LIN {X 0,Y 82.914,Z 593.303,A -85,B 0,C 180,E1 -30407.099,E2 -30407.099} C_VEL
LIN {X 0,Y 91.318,Z 585.109,A -85,B 0,C 180,E1 -30408.889,E2 -30408.889} C_VEL
LIN {X 0,Y 99.802,Z 575.115,A -85,B 0,C 180,E1 -30410.355,E2 -30410.355} C_VEL
LIN {X 0,Y 107.491,Z 563.809,A -85,B 0,C 180,E1 -30411.456,E2 -30411.456} C_VEL
LIN {X 0,Y 114.033,Z 551.61,A -85,B 0,C 180,E1 -30412.293,E2 -30412.293} C_VEL
LIN {X 0,Y 119.005,Z 539.43,A -85,B 0,C 180,E1 -30412.792,E2 -30412.792} C_VEL
LIN {X 0,Y 122.619,Z 526.994,A -85,B 0,C 180,E1 -30413.207,E2 -30413.207} C_VEL
LIN {X 0,Y 122.694,Z 526.451,A -85,B 0,C 180,E1 -30413.422,E2 -30413.422} C_VEL
LIN {X 0,Y 122.556,Z 525.141,A -85,B 0,C 180,E1 -30415.478,E2 -30415.478} C_VEL
LIN {X 0,Y 122.565,Z 523.201,A -85,B 0,C 180,E1 -30420,E2 -30420} C_VEL
LIN {X 0,Y 122.551,Z 525.424,A -85,B 0,C 180,E1 -30425.554,E2 -30425.554} C_VEL
LIN {X 0,Y 122.631,Z 526.514,A -85,B 0,C 180,E1 -30427.085,E2 -30427.085} C_VEL
LIN {X 0,Y 119.046,Z 538.887,A -85,B 0,C 180,E1 -30427.632,E2 -30427.632} C_VEL
LIN {X 0,Y 114.177,Z 550.868,A -85,B 0,C 180,E1 -30428.279,E2 -30428.279} C_VEL
LIN {X 0,Y 107.695,Z 563.005,A -85,B 0,C 180,E1 -30429.238,E2 -30429.238} C_VEL
LIN {X 0,Y 100.063,Z 574.276,A -85,B 0,C 180,E1 -30430.489,E2 -30430.489} C_VEL
LIN {X 0,Y 91.356,Z 584.529,A -85,B 0,C 180,E1 -30432.152,E2 -30432.152} C_VEL
LIN {X 0,Y 87.175,Z 588.67,A -85,B 0,C 180,E1 -30432.621,E2 -30432.621} C_VEL
LIN {X 0,Y 79.586,Z 595.067,A -85,B 0,C 180,E1 -30432.363,E2 -30432.363} C_VEL
LIN {X 0,Y 71.531,Z 600.835,A -85,B 0,C 180,E1 -30432.172,E2 -30432.172} C_VEL
LIN {X 0,Y 66.625,Z 603.967,A -85,B 0,C 180,E1 -30432.991,E2 -30432.991} C_VEL
LIN {X 0,Y 58.426,Z 608.742,A -85,B 0,C 180,E1 -30435.785,E2 -30435.785} C_VEL
LIN {X 0,Y 48.676,Z 613.433,A -85,B 0,C 180,E1 -30440.205,E2 -30440.205} C_VEL
LIN {X 0,Y 39.401,Z 617.015,A -85,B 0,C 180,E1 -30446.896,E2 -30446.896} C_VEL
LIN {X 0,Y 33.637,Z 618.862,A -85,B 0,C 180,E1 -30453.309,E2 -30453.309} C_VEL
LIN {X 0,Y 28.389,Z 620.248,A -85,B 0,C 180,E1 -30462.044,E2 -30462.044} C_VEL
LIN {X 0,Y 21.1,Z 621.833,A -85,B 0,C 180,E1 -30490.548,E2 -30490.548} C_VEL
LIN {X 0,Y 20.153,Z 622.053,A -85,B 0,C 180,E1 -30510.004,E2 -30510.004} C_VEL
LIN {X 0,Y 21.101,Z 621.857,A -85,B 0,C 180,E1 -30529.459,E2 -30529.459} C_VEL
LIN {X 0,Y 28.389,Z 620.301,A -85,B 0,C 180,E1 -30557.964,E2 -30557.964} C_VEL
LIN {X 0,Y 33.629,Z 618.939,A -85,B 0,C 180,E1 -30566.718,E2 -30566.718} C_VEL
LIN {X 0,Y 42.388,Z 616.065,A -85,B 0,C 180,E1 -30575.777,E2 -30575.777} C_VEL
LIN {X 0,Y 51.868,Z 612.161,A -85,B 0,C 180,E1 -30581.536,E2 -30581.536} C_VEL
LIN {X 0,Y 61.711,Z 607.122,A -85,B 0,C 180,E1 -30585.478,E2 -30585.478} C_VEL
LIN {X 0,Y 71.724,Z 600.776,A -85,B 0,C 180,E1 -30588.489,E2 -30588.489} C_VEL
LIN {X 0,Y 81.857,Z 592.844,A -85,B 0,C 180,E1 -30590.889,E2 -30590.889} C_VEL
LIN {X 0,Y 90.404,Z 584.751,A -85,B 0,C 180,E1 -30592.397,E2 -30592.397} C_VEL
LIN {X 0,Y 99.006,Z 574.873,A -85,B 0,C 180,E1 -30593.627,E2 -30593.627} C_VEL
LIN {X 0,Y 105.908,Z 565.141,A -85,B 0,C 180,E1 -30594.508,E2 -30594.508} C_VEL
LIN {X 0,Y 111.969,Z 554.581,A -85,B 0,C 180,E1 -30595.174,E2 -30595.174} C_VEL
LIN {X 0,Y 117.484,Z 542.178,A -85,B 0,C 180,E1 -30595.75,E2 -30595.75} C_VEL
LIN {X 0,Y 120.918,Z 531.884,A -85,B 0,C 180,E1 -30596.19,E2 -30596.19} C_VEL
LIN {X 0,Y 121.07,Z 530.606,A -85,B 0,C 180,E1 -30600,E2 -30600} C_VEL
LIN {X 0,Y 120.958,Z 531.95,A -85,B 0,C 180,E1 -30603.518,E2 -30603.518} C_VEL
LIN {X 0,Y 116.623,Z 544.629,A -85,B 0,C 180,E1 -30603.898,E2 -30603.898} C_VEL
LIN {X 0,Y 111.022,Z 556.642,A -85,B 0,C 180,E1 -30604.412,E2 -30604.412} C_VEL
LIN {X 0,Y 104.067,Z 568.172,A -85,B 0,C 180,E1 -30605.036,E2 -30605.036} C_VEL
LIN {X 0,Y 96.264,Z 578.56,A -85,B 0,C 180,E1 -30605.873,E2 -30605.873} C_VEL
LIN {X 0,Y 88.501,Z 587.056,A -85,B 0,C 180,E1 -30606.943,E2 -30606.943} C_VEL
LIN {X 0,Y 78.201,Z 596.263,A -85,B 0,C 180,E1 -30608.658,E2 -30608.658} C_VEL
LIN {X 0,Y 68.017,Z 603.672,A -85,B 0,C 180,E1 -30610.998,E2 -30610.998} C_VEL
LIN {X 0,Y 58.02,Z 609.627,A -85,B 0,C 180,E1 -30614.286,E2 -30614.286} C_VEL
LIN {X 0,Y 48.239,Z 614.33,A -85,B 0,C 180,E1 -30618.732,E2 -30618.732} C_VEL
LIN {X 0,Y 38.876,Z 617.925,A -85,B 0,C 180,E1 -30625.32,E2 -30625.32} C_VEL
LIN {X 0,Y 33.022,Z 619.778,A -85,B 0,C 180,E1 -30631.64,E2 -30631.64} C_VEL
LIN {X 0,Y 23.519,Z 622.171,A -85,B 0,C 180,E1 -30653.294,E2 -30653.294} C_VEL
LIN {X 0,Y 20.748,Z 622.783,A -85,B 0,C 180,E1 -30670.196,E2 -30670.196} C_VEL
LIN {X 0,Y 19.968,Z 622.998,A -85,B 0,C 180,E1 -30689.996,E2 -30689.996} C_VEL
LIN {X 0,Y 20.747,Z 622.762,A -85,B 0,C 180,E1 -30709.797,E2 -30709.797} C_VEL
LIN {X 0,Y 27.808,Z 621.124,A -85,B 0,C 180,E1 -30739.302,E2 -30739.302} C_VEL
LIN {X 0,Y 33.019,Z 619.708,A -85,B 0,C 180,E1 -30748.36,E2 -30748.36} C_VEL
LIN {X 0,Y 41.939,Z 616.756,A -85,B 0,C 180,E1 -30757.169,E2 -30757.169} C_VEL
LIN {X 0,Y 51.476,Z 612.766,A -85,B 0,C 180,E1 -30762.879,E2 -30762.879} C_VEL
LIN {X 0,Y 62.803,Z 606.729,A -85,B 0,C 180,E1 -30767.517,E2 -30767.517} C_VEL
LIN {X 0,Y 73.089,Z 599.938,A -85,B 0,C 180,E1 -30770.264,E2 -30770.264} C_VEL
LIN {X 0,Y 83.334,Z 591.643,A -85,B 0,C 180,E1 -30772.275,E2 -30772.275} C_VEL
LIN {X 0,Y 91.939,Z 583.13,A -85,B 0,C 180,E1 -30773.584,E2 -30773.584} C_VEL
LIN {X 0,Y 100.593,Z 572.617,A -85,B 0,C 180,E1 -30774.613,E2 -30774.613} C_VEL
LIN {X 0,Y 107.539,Z 562.211,A -85,B 0,C 180,E1 -30775.296,E2 -30775.296} C_VEL
LIN {X 0,Y 113.652,Z 550.719,A -85,B 0,C 180,E1 -30775.865,E2 -30775.865} C_VEL
LIN {X 0,Y 118.471,Z 538.818,A -85,B 0,C 180,E1 -30776.212,E2 -30776.212} C_VEL
LIN {X 0,Y 120.685,Z 531.737,A -85,B 0,C 180,E1 -30776.469,E2 -30776.469} C_VEL
LIN {X 0,Y 120.828,Z 530.26,A -85,B 0,C 180,E1 -30780,E2 -30780} C_VEL
LIN {X 0,Y 120.635,Z 531.717,A -85,B 0,C 180,E1 -30783.953,E2 -30783.953} C_VEL
LIN {X 0,Y 116.344,Z 544.263,A -85,B 0,C 180,E1 -30784.417,E2 -30784.417} C_VEL
LIN {X 0,Y 111.109,Z 555.609,A -85,B 0,C 180,E1 -30784.978,E2 -30784.978} C_VEL
LIN {X 0,Y 104.189,Z 567.217,A -85,B 0,C 180,E1 -30785.766,E2 -30785.766} C_VEL
LIN {X 0,Y 96.43,Z 577.65,A -85,B 0,C 180,E1 -30786.78,E2 -30786.78} C_VEL
LIN {X 0,Y 88.707,Z 586.174,A -85,B 0,C 180,E1 -30787.973,E2 -30787.973} C_VEL
LIN {X 0,Y 80.169,Z 594.029,A -85,B 0,C 180,E1 -30789.523,E2 -30789.523} C_VEL
LIN {X 0,Y 70.069,Z 601.693,A -85,B 0,C 180,E1 -30792.06,E2 -30792.06} C_VEL
LIN {X 0,Y 66.625,Z 603.967,A -85,B 0,C 180,E1 -30792.991,E2 -30792.991} C_VEL
LIN {X 0,Y 61.58,Z 606.937,A -85,B 0,C 180,E1 -30793.946,E2 -30793.946} C_VEL
LIN {X 0,Y 52.651,Z 611.259,A -85,B 0,C 180,E1 -30794.024,E2 -30794.024} C_VEL
LIN {X 0,Y 43.448,Z 614.93,A -85,B 0,C 180,E1 -30794.239,E2 -30794.239} C_VEL
LIN {X 0,Y 38.01,Z 616.77,A -85,B 0,C 180,E1 -30796.127,E2 -30796.127} C_VEL
LIN {X 0,Y 30.317,Z 619.031,A -85,B 0,C 180,E1 -30801.995,E2 -30801.995} C_VEL
LIN {X 0,Y 24.208,Z 620.416,A -85,B 0,C 180,E1 -30809.435,E2 -30809.435} C_VEL
LIN {X 0,Y 14.59,Z 622.001,A -85,B 0,C 180,E1 -30841.21,E2 -30841.21} C_VEL
LIN {X 0,Y 13.051,Z 622.22,A -85,B 0,C 180,E1 -30870.006,E2 -30870.006} C_VEL
LIN {X 0,Y 14.592,Z 622.024,A -85,B 0,C 180,E1 -30898.799,E2 -30898.799} C_VEL
LIN {X 0,Y 24.208,Z 620.468,A -85,B 0,C 180,E1 -30930.576,E2 -30930.576} C_VEL
LIN {X 0,Y 30.312,Z 619.106,A -85,B 0,C 180,E1 -30938.043,E2 -30938.043} C_VEL
LIN {X 0,Y 39.999,Z 616.232,A -85,B 0,C 180,E1 -30945.111,E2 -30945.111} C_VEL
LIN {X 0,Y 50.073,Z 612.327,A -85,B 0,C 180,E1 -30949.271,E2 -30949.271} C_VEL
LIN {X 0,Y 60.322,Z 607.288,A -85,B 0,C 180,E1 -30952.033,E2 -30952.033} C_VEL
LIN {X 0,Y 71.596,Z 600.267,A -85,B 0,C 180,E1 -30954.366,E2 -30954.366} C_VEL
LIN {X 0,Y 81.035,Z 593.009,A -85,B 0,C 180,E1 -30955.859,E2 -30955.859} C_VEL
LIN {X 0,Y 89.741,Z 584.915,A -85,B 0,C 180,E1 -30956.896,E2 -30956.896} C_VEL
LIN {X 0,Y 98.471,Z 575.036,A -85,B 0,C 180,E1 -30957.728,E2 -30957.728} C_VEL
LIN {X 0,Y 106.343,Z 563.897,A -85,B 0,C 180,E1 -30958.379,E2 -30958.379} C_VEL
LIN {X 0,Y 113.154,Z 551.609,A -85,B 0,C 180,E1 -30958.922,E2 -30958.922} C_VEL
LIN {X 0,Y 118.05,Z 540.074,A -85,B 0,C 180,E1 -30959.253,E2 -30959.253} C_VEL
LIN {X 0,Y 118.638,Z 538.372,A -85,B 0,C 180,E1 -30959.307,E2 -30959.307} C_VEL
LIN {X 0,Y 118.938,Z 537.482,A -85,B 0,C 180,E1 -30959.577,E2 -30959.577} C_VEL
LIN {X 0,Y 118.928,Z 537.521,A -85,B 0,C 180,E1 -30960,E2 -30960} C_VEL
LIN {X 0,Y 118.663,Z 538.323,A -85,B 0,C 180,E1 -30960.282,E2 -30960.282} C_VEL
LIN {X 0,Y 113.841,Z 550.25,A -85,B 0,C 180,E1 -30960.588,E2 -30960.588} C_VEL
LIN {X 0,Y 107.194,Z 562.581,A -85,B 0,C 180,E1 -30960.947,E2 -30960.947} C_VEL
LIN {X 0,Y 99.302,Z 574.069,A -85,B 0,C 180,E1 -30961.403,E2 -30961.403} C_VEL
LIN {X 0,Y 91.421,Z 583.316,A -85,B 0,C 180,E1 -30961.99,E2 -30961.99} C_VEL
LIN {X 0,Y 82.683,Z 591.755,A -85,B 0,C 180,E1 -30962.849,E2 -30962.849} C_VEL
LIN {X 0,Y 72.229,Z 600,A -85,B 0,C 180,E1 -30964.16,E2 -30964.16} C_VEL
LIN {X 0,Y 61.837,Z 606.651,A -85,B 0,C 180,E1 -30966.029,E2 -30966.029} C_VEL
LIN {X 0,Y 49.851,Z 612.733,A -85,B 0,C 180,E1 -30969.29,E2 -30969.29} C_VEL
LIN {X 0,Y 39.724,Z 616.687,A -85,B 0,C 180,E1 -30973.319,E2 -30973.319} C_VEL
LIN {X 0,Y 29.904,Z 619.611,A -85,B 0,C 180,E1 -30979.926,E2 -30979.926} C_VEL
LIN {X 0,Y 18.315,Z 622.004,A -85,B 0,C 180,E1 -30999.865,E2 -30999.865} C_VEL
LIN {X 0,Y 14.253,Z 622.616,A -85,B 0,C 180,E1 -31020.449,E2 -31020.449} C_VEL
LIN {X 0,Y 12.865,Z 622.83,A -85,B 0,C 180,E1 -31049.994,E2 -31049.994} C_VEL
LIN {X 0,Y 14.252,Z 622.594,A -85,B 0,C 180,E1 -31079.541,E2 -31079.541} C_VEL
LIN {X 0,Y 23.783,Z 620.956,A -85,B 0,C 180,E1 -31112.434,E2 -31112.434} C_VEL
LIN {X 0,Y 29.901,Z 619.54,A -85,B 0,C 180,E1 -31120.075,E2 -31120.075} C_VEL
LIN {X 0,Y 39.721,Z 616.587,A -85,B 0,C 180,E1 -31126.684,E2 -31126.684} C_VEL
LIN {X 0,Y 49.847,Z 612.597,A -85,B 0,C 180,E1 -31130.722,E2 -31130.722} C_VEL
LIN {X 0,Y 61.656,Z 606.56,A -85,B 0,C 180,E1 -31133.997,E2 -31133.997} C_VEL
LIN {X 0,Y 72.226,Z 599.768,A -85,B 0,C 180,E1 -31135.84,E2 -31135.84} C_VEL
LIN {X 0,Y 82.679,Z 591.474,A -85,B 0,C 180,E1 -31137.166,E2 -31137.166} C_VEL
LIN {X 0,Y 91.418,Z 582.96,A -85,B 0,C 180,E1 -31138.019,E2 -31138.019} C_VEL
LIN {X 0,Y 100.175,Z 572.446,A -85,B 0,C 180,E1 -31138.668,E2 -31138.668} C_VEL
LIN {X 0,Y 108.067,Z 560.606,A -85,B 0,C 180,E1 -31139.13,E2 -31139.13} C_VEL
LIN {X 0,Y 113.978,Z 549.173,A -85,B 0,C 180,E1 -31139.487,E2 -31139.487} C_VEL
LIN {X 0,Y 118.388,Z 538.126,A -85,B 0,C 180,E1 -31139.661,E2 -31139.661} C_VEL
LIN {X 0,Y 118.698,Z 537.187,A -85,B 0,C 180,E1 -31140,E2 -31140} C_VEL
LIN {X 0,Y 118.716,Z 537.123,A -85,B 0,C 180,E1 -31140.424,E2 -31140.424} C_VEL
LIN {X 0,Y 118.143,Z 538.822,A -85,B 0,C 180,E1 -31140.788,E2 -31140.788} C_VEL
LIN {X 0,Y 113.084,Z 551.065,A -85,B 0,C 180,E1 -31141.138,E2 -31141.138} C_VEL
LIN {X 0,Y 106.344,Z 563.348,A -85,B 0,C 180,E1 -31141.689,E2 -31141.689} C_VEL
LIN {X 0,Y 99.348,Z 573.468,A -85,B 0,C 180,E1 -31142.276,E2 -31142.276} C_VEL
LIN {X 0,Y 91.489,Z 582.769,A -85,B 0,C 180,E1 -31143.009,E2 -31143.009} C_VEL
LIN {X 0,Y 82.78,Z 591.238,A -85,B 0,C 180,E1 -31143.999,E2 -31143.999} C_VEL
LIN {X 0,Y 73.1,Z 598.969,A -85,B 0,C 180,E1 -31145.517,E2 -31145.517} C_VEL
LIN {X 0,Y 63.761,Z 605.108,A -85,B 0,C 180,E1 -31147.249,E2 -31147.249} C_VEL
LIN {X 0,Y 53.487,Z 610.599,A -85,B 0,C 180,E1 -31149.783,E2 -31149.783} C_VEL
LIN {X 0,Y 43.333,Z 614.908,A -85,B 0,C 180,E1 -31153.324,E2 -31153.324} C_VEL
LIN {X 0,Y 38.01,Z 616.77,A -85,B 0,C 180,E1 -31156.127,E2 -31156.127} C_VEL
LIN {X 0,Y 32.551,Z 618.379,A -85,B 0,C 180,E1 -31158.713,E2 -31158.713} C_VEL
LIN {X 0,Y 22.952,Z 620.494,A -85,B 0,C 180,E1 -31161.4,E2 -31161.4} C_VEL
LIN {X 0,Y 15.163,Z 621.634,A -85,B 0,C 180,E1 -31165.259,E2 -31165.259} C_VEL
LIN {X 0,Y 9.716,Z 622.121,A -85,B 0,C 180,E1 -31176.18,E2 -31176.18} C_VEL
LIN {X 0,Y 8.203,Z 622.204,A -85,B 0,C 180,E1 -31184.353,E2 -31184.353} C_VEL
LIN {X 0,Y 5.958,Z 622.387,A -85,B 0,C 180,E1 -31230.013,E2 -31230.013} C_VEL
LIN {X 0,Y 9.044,Z 622.191,A -85,B 0,C 180,E1 -31281.01,E2 -31281.01} C_VEL
LIN {X 0,Y 21.621,Z 620.635,A -85,B 0,C 180,E1 -31307.216,E2 -31307.216} C_VEL
LIN {X 0,Y 28.428,Z 619.273,A -85,B 0,C 180,E1 -31311.463,E2 -31311.463} C_VEL
LIN {X 0,Y 38.785,Z 616.398,A -85,B 0,C 180,E1 -31315.31,E2 -31315.31} C_VEL
LIN {X 0,Y 49.248,Z 612.493,A -85,B 0,C 180,E1 -31317.414,E2 -31317.414} C_VEL
LIN {X 0,Y 56.248,Z 609.255,A -85,B 0,C 180,E1 -31318.382,E2 -31318.382} C_VEL
LIN {X 0,Y 56.581,Z 609.11,A -85,B 0,C 180,E1 -31320,E2 -31320} C_VEL
LIN {X 0,Y 45.701,Z 613.998,A -85,B 0,C 180,E1 -31321.581,E2 -31321.581} C_VEL
LIN {X 0,Y 35.222,Z 617.592,A -85,B 0,C 180,E1 -31323.882,E2 -31323.882} C_VEL
LIN {X 0,Y 28.28,Z 619.444,A -85,B 0,C 180,E1 -31326.225,E2 -31326.225} C_VEL
LIN {X 0,Y 14.795,Z 621.837,A -85,B 0,C 180,E1 -31338.171,E2 -31338.171} C_VEL
LIN {X 0,Y 8.797,Z 622.449,A -85,B 0,C 180,E1 -31356.959,E2 -31356.959} C_VEL
LIN {X 0,Y 5.754,Z 622.663,A -85,B 0,C 180,E1 -31409.987,E2 -31409.987} C_VEL
LIN {X 0,Y 8.795,Z 622.427,A -85,B 0,C 180,E1 -31463.031,E2 -31463.031} C_VEL
LIN {X 0,Y 21.433,Z 620.787,A -85,B 0,C 180,E1 -31489.627,E2 -31489.627} C_VEL
LIN {X 0,Y 28.277,Z 619.371,A -85,B 0,C 180,E1 -31493.777,E2 -31493.777} C_VEL
LIN {X 0,Y 38.706,Z 616.418,A -85,B 0,C 180,E1 -31497.001,E2 -31497.001} C_VEL
LIN {X 0,Y 51.829,Z 611.234,A -85,B 0,C 180,E1 -31499.345,E2 -31499.345} C_VEL
LIN {X 0,Y 56.223,Z 609.119,A -85,B 0,C 180,E1 -31500,E2 -31500} C_VEL
LIN {X 0,Y 56.248,Z 609.079,A -85,B 0,C 180,E1 -31501.704,E2 -31501.704} C_VEL
LIN {X 0,Y 45.755,Z 613.769,A -85,B 0,C 180,E1 -31503.271,E2 -31503.271} C_VEL
LIN {X 0,Y 35.32,Z 617.352,A -85,B 0,C 180,E1 -31505.803,E2 -31505.803} C_VEL
LIN {X 0,Y 28.429,Z 619.199,A -85,B 0,C 180,E1 -31508.584,E2 -31508.584} C_VEL
LIN {X 0,Y 15.013,Z 621.567,A -85,B 0,C 180,E1 -31520.581,E2 -31520.581} C_VEL
LIN {X 0,Y 8.203,Z 622.204,A -85,B 0,C 180,E1 -31544.353,E2 -31544.353} C_VEL
LIN {X 0,Y 8.203,Z 622.204,A -85,B 0,C 180,E1 -31544.353,E2 -31544.353}

QRS_NEXT_CUT()

QRS_NEXT()
QRS_HOME()

END
